// TIA Portal V18 export
TYPE "AGV_ShW"
// stored: IsFailsafeCompliant false
   STRUCT
      Trigger : Bool;
      Result : Int;
      Completed : Bool;
      TaskNo : Int;   // 10:上料 20：下料 30：取空箱 40：补空箱
      PointName : String[48];
      materialLot : String[48];
      materialQuantity : Int;
      SafetySignal : Bool;   // 0：不安全 1： 安全
      ProcessBit : Bool;   // 0：可以继续发送请求 1：不能重新发送请求
   END_STRUCT;
END_TYPE
